# EPICS substitutions: edgeRoboArmIOC/support/xxx-5-6/iocBoot/iocLinux/substitutions/LogitechExtreme3DPro.substitutions
file "$(USB)/usbApp/Db/AnalogAxis.template"
{
pattern
{P     R               PARAM               PORT          FLNK}
{xxx:  A1:Vertical     VERTICAL_STATE      LOGITECH      xxx:A1:shoulder}
{xxx:  A1:Rotation     ROTATION_STATE      LOGITECH      xxx:A1:base}
{xxx:  A1:Switch       SWITCH_STATE        LOGITECH      xxx:A1:move_lock}
{xxx:  A1:Hat          HAT_STATE           LOGITECH      xxx:A1:wrist}
}

file "$(USB)/usbApp/Db/DigitalButton.template"
{
pattern
{P     R               PARAM               PORT          FLNK}
{xxx:  A1:Trigger      TRIGGER_PRESSED     LOGITECH      xxx:A1:grip}
{xxx:  A1:LButton      LBUTTON_PRESSED     LOGITECH      xxx:A1:grip}
{xxx:  A1:Button3      BUTTON3_PRESSED     LOGITECH      xxx:A1:elbow}
{xxx:  A1:Button5      BUTTON5_PRESSED     LOGITECH      xxx:A1:elbow}
{xxx:  A1:Button11     BUTTON11_PRESSED    LOGITECH      xxx:A1:led}
}

file "$(TOP)/iocBoot/$(IOC)/substitutions/AxisMove.template"
{
pattern
{P     R               LOCK               AXIS             DEAD_LOW   DEAD_HIGH   OUT}
{xxx:  A1:move_lock    0                  xxx:A1:Switch    0          126         ""}
{xxx:  A1:base         xxx:A1:move_lock   xxx:A1:Rotation  50         200         xxx:A1:base_move}
{xxx:  A1:shoulder     xxx:A1:move_lock   xxx:A1:Vertical  50         600         xxx:A1:shoulder_move}
}

file "$(TOP)/iocBoot/$(IOC)/substitutions/ButtonMove.template"
{
pattern
{P     R                LOCK              BUTTONA            BUTTONB           OUT}
{xxx:  A1:led           0                 0                  xxx:A1:Button11   xxx:A1:led_onoff}
{xxx:  A1:elbow         xxx:A1:move_lock  xxx:A1:Button3     xxx:A1:Button5    xxx:A1:elbow_move}
{xxx:  A1:grip          xxx:A1:move_lock  xxx:A1:LButton     xxx:A1:Trigger    xxx:A1:grip_move}
}

file "$(TOP)/iocBoot/$(IOC)/substitutions/DiscreteMove.template"
{
pattern
{P     R                LOCK               AXIS            VALA    VALB     OUT}
{xxx:  A1:wrist         xxx:A1:move_lock   xxx:A1:Hat      4       0        xxx:A1:wrist_move}
}
